KUKA KRL program: end_weld_respot.src

&ACCESS RVP
&REL 6
&PARAM TEMPLATE = C:\KRC\Roboter\Template\ExpertVorgabe
&PARAM EDITMASK = *
DEF END_WELD_RESPOT( )


;FOLD ; SOLDA RESPOT FINALIZADA;%{PE}%R 4.1.16,%MKUKATPBASIS,%CCOMMENT,%VNORMAL,%P 2:SOLDA RESPOT FINALIZADA
;ENDFOLD
;FOLD PULSE 3334 'R1_Solda Respot OK' State=TRUE Time=3 sec;%{PE}%R 8.2.20,%MKUKATPBASIS,%COUT,%VPULSE,%P 2:3334, 3:R1_Solda Respot OK, 5:TRUE, 6:, 8:3
PULSE($OUT[3334], TRUE,3)
;ENDFOLD


END
